FUNCTION_BLOCK FB_HnhtCnLinkage
VAR_INPUT	
	//control struct for hnht cn linkage
	controlAutomatic : ST_HnhtCnLinkageControl;
END_VAR
VAR_OUTPUT
END_VAR
VAR
	//systems
	VentilationSystem : FB_VentilationSystem;
	
	//internal variables
	bAlgorithmPermission : BOOL;
	
	//PCM Supply System
	PCMSupplySystem : FB_PCMSupplySystem;
END_VAR

bAlgorithmPermission := controlAutomatic.bAlgorithmPermission_HNHT AND controlAutomatic.bAlgorithmPermission_CN;

//ventilation system has its own controller, only valves are controlled
VentilationSystem(bSetStatusOnAutomatic := TRUE,
	fSetPointAutomatic := 0,
	bAlgorithmPermission := bAlgorithmPermission,
	bHeatingModeAutomatic := controlAutomatic.bHeatingMode);

PCMSupplySystem(bSetStatusOnAutomatic := TRUE, 
	bAlgorithmPermission := bAlgorithmPermission,
	fSetPointAutomatic := 9);

END_FUNCTION_BLOCK

(* stored: Version 1.1.0.1, ProductVersion 3.1.4024.10
   POU FB_HnhtCnLinkage: Id {dda8ef66-5894-40a8-a8ba-58cd641df7f0}, SpecialFunc None *)
